// TIA Portal V18 export
DATA_BLOCK "DB_SideShifter_1"   // DB2
// stored: InstanceOfName SideShifter, InstanceOfType FB
"SideShifter"
   // VAR_INPUT
   //    Hydraulic_Up : Bool;
   //    Hydraulic_Down : Bool;
   //    Hydraulic_Unit : Bool;
   //    Homing1 : Bool;
   //    Homing2 : Bool;
   //    Homing3 : Bool;
   //    Safety : Bool;
   // END_VAR
   // VAR_OUTPUT
   //    Hydraulic_Actuator1_Up : Bool;
   //    Hydraulic_Actuator1_Down : Bool;
   //    Hydraulic_Actuator2_Up : Bool;
   //    Hydraulic_Actuator2_Down : Bool;
   //    Hydraulic_Unit1 : Bool;
   //    Hydraulic_Unit2 : Bool;
   // END_VAR
BEGIN
END_DATA_BLOCK
